FUNCTION_BLOCK TcoDesignerClearInspectionResults_v_2_x_x EXTENDS TcoCore.TcoTask
VAR_IN_OUT
	inoIoData	: TcoDesignerData_2_x_x;
    inoConfig	: TcoDesignerConfig_v_2_x_x;
	inoStatus	: TcoDesignerStatus_v_2_x_x;	
	//inoResults	: TcoInsightResults_v_5_x_x;
END_VAR
VAR
    {attribute 'hide'} 
	_progress : INT := 0;
    {attribute 'hide'} 
	_infoTimer :  TON;
    {attribute 'hide'} 
	_errorTimer :  TON;
    {attribute 'hide'} 
	_varInfo : __SYSTEM.VAR_INFO;
    {attribute 'hide'} 
	_sb : TcoCore.StringBuilder;
END_VAR

IF Execute() THEN
	IF _progress = 0 THEN
		IF NOT __ISVALIDREF(inoIoData) THEN
			_varInfo :=__VARINFO(inoIoData);
			Messenger.Programming(_sb.Clear().Append('<#Invalid reference: #>').Append(_varInfo.Symbol).ToString()).Pin();
		ELSIF NOT __ISVALIDREF(inoConfig) THEN                                                  
			_varInfo :=__VARINFO(inoConfig);                                                    
			Messenger.Programming(_sb.Clear().Append('<#Invalid reference: #>').Append(_varInfo.Symbol).ToString()).Pin();
		ELSIF NOT __ISVALIDREF(inoStatus) THEN                                                  
			_varInfo :=__VARINFO(inoStatus);                                                    
			Messenger.Programming(_sb.Clear().Append('<#Invalid reference: #>').Append(_varInfo.Symbol).ToString()).Pin();
//		ELSIF NOT __ISVALIDREF(inoResults) THEN                                              
//			_varInfo :=__VARINFO(inoResults);                                                
//			Messenger.Programming(_sb.Clear().Append('<#Invalid reference: #>').Append(_varInfo.Symbol).ToString()).Pin();
		ELSE
			_progress := _progress + 1;
		END_IF
	END_IF
	
	IF _progress = 1 THEN
		CallTimers(FALSE);
		THIS^.inoIoData.PlcToPc.Trigger := FALSE;
		THIS^.inoIoData.PlcToPc.LoadJob := FALSE;
		
		THIS^.inoIoData.PlcToPc.Reset := FALSE;
		THIS^.inoIoData.PlcToPc.ResultsAck := FALSE;

		THIS^.inoIoData.PlcToPc.ClearResults:=FALSE;

		_progress := _progress + 1;
	END_IF
	
	IF _progress = 2 THEN
		THIS^.Messenger.OnCondition(_infoTimer.Q).Info('<#Reset Request!#>'); 
		THIS^.inoIoData.PlcToPc.Reset := TRUE;
		IF THIS^.inoIoData.PcToPlc.InspectionReady
			AND NOT THIS^.inoIoData.PcToPlc.ClearResultsAck
			AND NOT THIS^.inoIoData.PcToPlc.ResultsAvailable 
			AND NOT THIS^.inoIoData.PcToPlc.JobLoadDone THEN
			THIS^.inoIoData.PlcToPc.Reset := FALSE;
			_progress := _progress + 1;
		END_IF
	END_IF
	
	IF _progress = 3 THEN
		THIS^.Messenger.OnCondition(_infoTimer.Q).Warning('<#Waiting for the Online signal!#>'); 
		IF THIS^.inoIoData.PcToPlc.SystemOnline THEN
			CallTimers(FALSE);
			_progress := _progress + 1;
		END_IF
	END_IF
	
	IF _progress = 4 THEN
		THIS^.Messenger.OnCondition(_infoTimer.Q).Info('<#Waiting to Acknowledge results!#>'); 
		THIS^.inoIoData.PlcToPc.ResultsAck:=TRUE;
		IF NOT THIS^.inoIoData.PcToPlc.ResultsAvailable  THEN
			THIS^.inoIoData.PlcToPc.ResultsAck:=FALSE;
			CallTimers(FALSE);
			_progress := _progress + 1;
		END_IF
	END_IF
	
	IF _progress = 5 THEN
		THIS^.Messenger.OnCondition(_infoTimer.Q).Info('<#Waiting to clear old data!#>'); 
		THIS^.inoIoData.PlcToPc.ClearResults:=TRUE;
	
		IF  THIS^.inoIoData.PcToPlc.ClearResultsAck  THEN
			THIS^.inoIoData.PlcToPc.ClearResults:=FALSE;
			CallTimers(FALSE);
			_progress := _progress + 1;
		END_IF
	END_IF
	
	IF _progress = 6 THEN
		THIS^.Messenger.OnCondition(_infoTimer.Q).Info('<#Waiting for Inspection ready!#>'); 
		IF THIS^.inoIoData.PcToPlc.InspectionReady 
			 THEN
			CallTimers(FALSE);
			_progress := _progress + 1;
		END_IF
	END_IF
	
	IF _progress = 7 THEN	
		THIS^.Messenger.OnCondition(_infoTimer.Q).Info('<#Waiting for data were cleared!#>'); 
			IF  NOT THIS^.inoIoData.PcToPlc.ClearResultsAck
			AND NOT THIS^.inoIoData.PcToPlc.InspectionResults.ResultFail
			AND NOT THIS^.inoIoData.PcToPlc.InspectionResults.ResultPass THEN
			CallTimers(FALSE);
			THIS^.DoneWhen(TRUE);
		END_IF
	END_IF
	
	CallTimers(TRUE);
	
		THIS^.ThrowWhen(_errorTimer.Q   OR THIS^.inoIoData.PcToPlc.Error );	
END_IF

METHOD CallTimers
VAR_INPUT
	inValue : BOOL;
END_VAR
IF  __ISVALIDREF(inoConfig) AND THIS^.inoConfig.ErrorTime <> T#0S OR NOT inValue THEN  
_errorTimer(IN := inValue, PT := THIS^.inoConfig.ErrorTime);
END_IF;
IF  __ISVALIDREF(inoConfig) AND THIS^.inoConfig.InfoTime <>T#0S OR NOT inValue THEN  
_infoTimer(IN := inValue, PT := THIS^.inoConfig.InfoTime);
END_IF;
END_METHOD

(*~
	<docu>
		<summary>
			Executes when task is aborted.
		</summary>			
	</docu>	
~*)
METHOD PROTECTED OnAbort
THIS^.inoStatus.ActionDescription := '<#Clearing of the inspection results aborted, while not yet finished.#>';
END_METHOD

(*~
	<docu>
		<summary>
			Executes when task reaches the ```Done``` state .
		</summary>			
	</docu>	
~*)
METHOD PROTECTED OnDone
THIS^.inoStatus.ActionDescription := '<#Clearing of the inspection results was completed succesfully.#>'; 
_progress:=0;
END_METHOD

(*~
	<docu>
		<summary>
			Executes when task reaches the ```Error``` state.
			<para>
				Do not confuse with <see cref="PlcDocu.TcoCore.TcoTask.WhileError()"/>, that is called cyclically until '''Error''' state is left.
			</para>
		</summary>			
	</docu>	
~*)
METHOD PROTECTED OnError
THIS^.inoStatus.ActionDescription := '<#Clearing of the inspection results finished with error.#>';
END_METHOD

METHOD PROTECTED OnStart
THIS^.inoStatus.ActionDescription := '<#Clearing of the inspection results started.#>';
END_METHOD

(*~
	<docu>
		<summary>
			Restores this instance to the Ready state. Can be called explicitly or from within one of the restore mechanisms.
			<para>
				See also <see cref="PlcDocu.TcoCore.TcoTask.AutoRestorable()"/>
			</para>
		</summary>			
	</docu>	
~*)
METHOD Restore : ITcoRestorable
SUPER^.Restore();
_progress := 0;
CallTimers(FALSE);
Messenger.UnPin();
END_METHOD

END_FUNCTION_BLOCK

(* stored: Version 1.1.0.1, ProductVersion 3.1.4024.12
   POU TcoDesignerClearInspectionResults_v_2_x_x: Id {e8ef7c4c-3177-0824-2334-795cb0911f81}, SpecialFunc None
   Method CallTimers: Id {20f1120c-e43e-0225-1470-baa6a7d49a9f}
   Method OnAbort: Id {eeeb0d6e-b9d5-027e-212b-c27a9bb61750}
   Method OnDone: Id {0c3f7c44-2320-0e67-0ddb-e2bff473064c}
   Method OnError: Id {20621a47-bfd9-03e5-3b6f-cd33eb6b89e9}
   Method OnStart: Id {7c61dc07-cfb4-0703-05b6-4b1966f1999e}
   Method Restore: Id {ef084e57-b0bb-067b-3024-acafaa2e17dc} *)
